INTERFACE I_HostErrors EXTENDS __SYSTEM.IQueryInterface

METHOD AddError
VAR_INPUT
	Error : I_Error;
END_VAR
END_METHOD

PROPERTY PUBLIC HasRaisedError : BOOL
GET
END_GET
END_PROPERTY

END_INTERFACE

(* stored: Version 1.1.0.1, ProductVersion 3.1.4024.12
   Itf I_HostErrors: Id {6c14ee43-6ab7-0c30-3bf7-4a331785d2fc}
   Method AddError: Id {23aee699-1229-0461-1c27-f5ff339c8835}
   Property HasRaisedError: Id {89f3b71d-f74d-4e4e-b2e3-984400e16d37}
   Get Get: Id {d76a8ec5-a42a-4c96-8539-f71507e247fc} *)
